TYPE Example2WrappedComponents_Control EXTENDS TcoCore.TcoStruct:
STRUCT

		Setpoint1:INT;
		Up:BOOL;
		CommandAscii:STRING;
END_STRUCT
END_TYPE

(* stored: Version 1.1.0.1
   DUT Example2WrappedComponents_Control: Id {522653ec-0163-04ff-3aa5-9302596f169e} *)
